// TIA Portal V19 export
FUNCTION_BLOCK "TYPIC_C103_IF_OVB"   // FB32, FBD
TITLE = TYPIC_C103_IF_OVB: LSBB
{ S7_Optimized_Access := 'TRUE' }
AUTHOR : OCOTECH
FAMILY : Typical
NAME : C103.705
// Logisch Object Besturing: C103.805
// 
// De interne functie laagspanningsverdeelbord buiten verzorgt de bewaking van een laagspanningsverdeelbord buiten.
// stored: MemoryReserve 10, SetENOAutomatically false
   VAR_INPUT
      EXT_AUT { ExternalAccessible := 'False'; ExternalVisible := 'False'; ExternalWritable := 'False'} : Bool;   // Externe (hoofd) beveiliging (1 = OK)
      EXT_HW { ExternalAccessible := 'False'; ExternalVisible := 'False'; ExternalWritable := 'False'} : Bool;   // Sturings hardware (PLC) bewaking (1 = OK)
      IN_SCL { ExternalAccessible := 'False'; ExternalVisible := 'False'; ExternalWritable := 'False'} : Bool;   // LSB ingangszone 400V/230V
   END_VAR
   VAR_OUTPUT
      VAR_IF_OVB { ExternalAccessible := 'False'; ExternalVisible := 'False'; ExternalWritable := 'False'} : "C103_VAR_IF_OVB_TYPIC";   // Struct met alle variabelen naar bovenliggende functies
   END_VAR
   VAR
      STO { ExternalWritable := 'False'} : Struct   // Storingen
         A001 { ExternalAccessible := 'False'; ExternalVisible := 'False'} : Bool;   // Laagspanningsverdeelbord buiten beveiliging aangesproken
         A002 { ExternalAccessible := 'False'; ExternalVisible := 'False'} : Bool;   // Laagspanningsverdeelbord buiten in dienstkoker in storing
      END_STRUCT;
      VAR { ExternalWritable := 'False'} : Struct   // Variabelen
         SCL { ExternalAccessible := 'False'; ExternalVisible := 'False'} : Bool;   // Standmelding ingangszone 400V/230V
      END_STRUCT;
   END_VAR
BEGIN

REGION Network 1: START
END_REGION

REGION Network 2: +++ Verwerking meetwaarden en statussen +++
   // De meetwaarde en status wordt ontvangen vanuit de interne sturing.
END_REGION

REGION Network 3: +++ Storingen +++
   // Combinatie van de storingen
END_REGION

REGION Network 4: Storing A001: Laagspanningsverdeelbord buiten beveiliging aangesproken
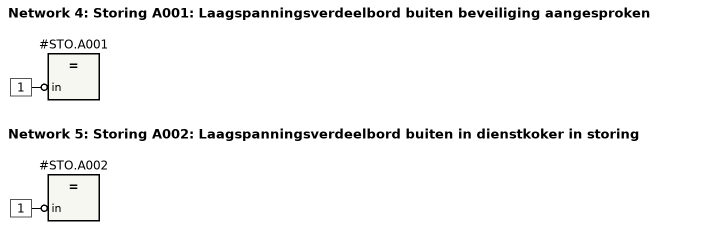
   #STO.A001 := NOT 1;
END_REGION

REGION Network 5: Storing A002: Laagspanningsverdeelbord buiten in dienstkoker in storing
   #STO.A002 := NOT 1;
END_REGION

REGION Network 6 (SCL): EINDE
   // Variabelen van intern scada rakvlak naar outputs copieren
   #VAR_IF_OVB.SCL := #VAR.SCL;
END_REGION
END_FUNCTION_BLOCK
